FUNCTION_BLOCK UA_NodeReleaseHandleWrapper IMPLEMENTS I_OPCUA_NodeReleaseHandle
VAR_INPUT
END_VAR
VAR_OUTPUT
END_VAR
VAR
	uaNodeReleaseHandle : UA_NodeReleaseHandle;
END_VAR

{warning 'add method implementation '}
METHOD start : BOOL
VAR_INPUT
	Execute	: BOOL;
	ConnectionHdl	: DWORD;
	NodeHdl	: DWORD;
	Timeout	: TIME := DEFAULT_ADS_TIMEOUT;
END_VAR
VAR_OUTPUT
	Done	: BOOL;
	Busy	: BOOL;
	Error	: BOOL;
	ErrorID	: DWORD;
END_VAR
uaNodeReleasehandle(Execute := execute, 
					connectionhdl := connectionhdl, 
					nodehdl := nodehdl, 
					timeout := timeout,
					Done => Done,
					Busy => Busy,
					Error => Error,
					ErrorID => ErrorID);
END_METHOD

END_FUNCTION_BLOCK

(* stored: Version 1.1.0.1, ProductVersion 3.1.4024.9
   POU UA_NodeReleaseHandleWrapper: Id {6d74129d-b57f-4042-be40-2550de29caa1}, SpecialFunc None
   Method start: Id {fc24c77a-3fe1-461f-81af-799c6aba19c7} *)
